// TIA Portal V19 export
FUNCTION "FC40_MasterComm" : Void   // FC40, LAD
{ S7_Optimized_Access := 'TRUE' }
// stored: AutoNumber false, IsIECCheckEnabled true, SetENOAutomatically true
BEGIN

REGION Network 1: Master Communication
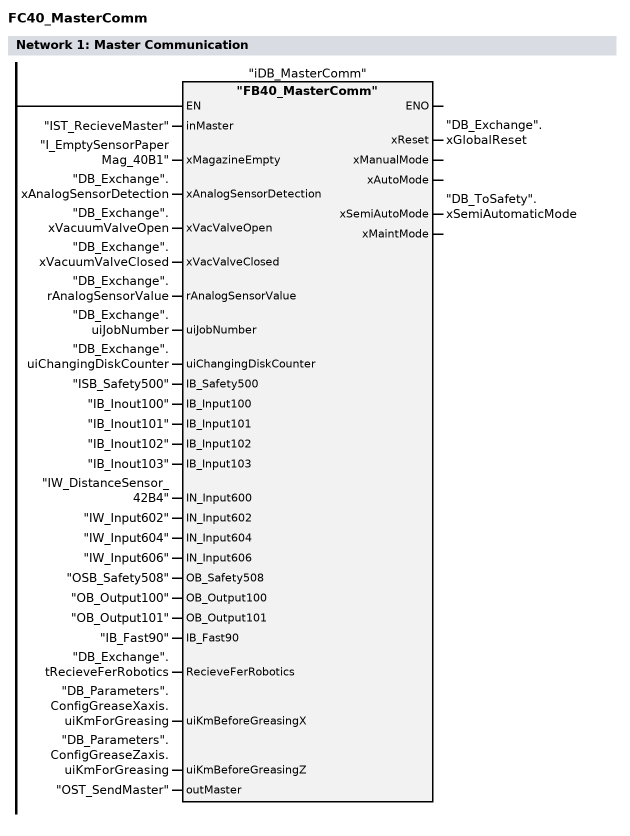
   RUNG wire#powerrail
      "iDB_MasterComm"(inMaster := "IST_RecieveMaster", xMagazineEmpty := "I_EmptySensorPaperMag_40B1", xAnalogSensorDetection := "DB_Exchange".xAnalogSensorDetection, xVacValveOpen := "DB_Exchange".xVacuumValveOpen, xVacValveClosed := "DB_Exchange".xVacuumValveClosed, rAnalogSensorValue := "DB_Exchange".rAnalogSensorValue, uiJobNumber := "DB_Exchange".uiJobNumber, uiChangingDiskCounter := "DB_Exchange".uiChangingDiskCounter, IB_Safety500 := "ISB_Safety500", IB_Input100 := "IB_Inout100", IB_Input101 := "IB_Inout101", IB_Input102 := "IB_Inout102", IB_Input103 := "IB_Inout103", IN_Input600 := "IW_DistanceSensor_42B4", IN_Input602 := "IW_Input602", IN_Input604 := "IW_Input604", IN_Input606 := "IW_Input606", OB_Safety508 := "OSB_Safety508", OB_Output100 := "OB_Output100", OB_Output101 := "OB_Output101", IB_Fast90 := "IB_Fast90", RecieveFerRobotics := "DB_Exchange".tRecieveFerRobotics, uiKmBeforeGreasingX := "DB_Parameters".ConfigGreaseXaxis.uiKmForGreasing, uiKmBeforeGreasingZ := "DB_Parameters".ConfigGreaseZaxis.uiKmForGreasing, outMaster := "OST_SendMaster", xReset => "DB_Exchange".xGlobalReset, xManualMode =>, xAutoMode =>, xSemiAutoMode => "DB_ToSafety".xSemiAutomaticMode, xMaintMode =>)
   END_RUNG
   // the same network as SCL:
   "iDB_MasterComm"(inMaster := "IST_RecieveMaster",   // "FB40_MasterComm"
                    xMagazineEmpty := "I_EmptySensorPaperMag_40B1",
                    xAnalogSensorDetection := "DB_Exchange".xAnalogSensorDetection,
                    xVacValveOpen := "DB_Exchange".xVacuumValveOpen,
                    xVacValveClosed := "DB_Exchange".xVacuumValveClosed,
                    rAnalogSensorValue := "DB_Exchange".rAnalogSensorValue,
                    uiJobNumber := "DB_Exchange".uiJobNumber,
                    uiChangingDiskCounter := "DB_Exchange".uiChangingDiskCounter,
                    IB_Safety500 := "ISB_Safety500",
                    IB_Input100 := "IB_Inout100",
                    IB_Input101 := "IB_Inout101",
                    IB_Input102 := "IB_Inout102",
                    IB_Input103 := "IB_Inout103",
                    IN_Input600 := "IW_DistanceSensor_42B4",
                    IN_Input602 := "IW_Input602",
                    IN_Input604 := "IW_Input604",
                    IN_Input606 := "IW_Input606",
                    OB_Safety508 := "OSB_Safety508",
                    OB_Output100 := "OB_Output100",
                    OB_Output101 := "OB_Output101",
                    IB_Fast90 := "IB_Fast90",
                    RecieveFerRobotics := "DB_Exchange".tRecieveFerRobotics,
                    uiKmBeforeGreasingX := "DB_Parameters".ConfigGreaseXaxis.uiKmForGreasing,
                    uiKmBeforeGreasingZ := "DB_Parameters".ConfigGreaseZaxis.uiKmForGreasing,
                    outMaster := "OST_SendMaster",
                    xReset => "DB_Exchange".xGlobalReset,
                    xSemiAutoMode => "DB_ToSafety".xSemiAutomaticMode);
END_REGION
END_FUNCTION
